(* PLC project Sin nombre, Desconocido Sin nombre 1 *)
(* stored: creationDateTime 2024-04-02T14:40:19, modificationDateTime 2024-04-04T08:12:00 *)

PROGRAM program0
  VAR
    START AT %IX0.0 : BOOL;
    STOP AT %IX0.1 : BOOL;
    INPUT0 AT %IX0.2 : BOOL := TRUE;
    OUTPUT0 AT %QX0.0 : BOOL;
    OUTPUT1 AT %QX0.1 : BOOL;
    STOP_LIGHT AT %QX0.2 : BOOL;
    START_LIGHT AT %QX0.3 : BOOL;
  END_VAR
  VAR
    IR1 : BOOL;
    IR2 : BOOL;
    IR3 : BOOL;
    IR4 : BOOL;
    IR5 : BOOL;
    TON_TIME1 : TIME := T#5S;
    COUNT_START : INT := 5;
    TON0 : TON;
    CTU0 : CTU;
  END_VAR
  VAR  (* added by the conversion: wires and edge detectors of the diagram *)
    R_TRIG1 : R_TRIG;
  END_VAR

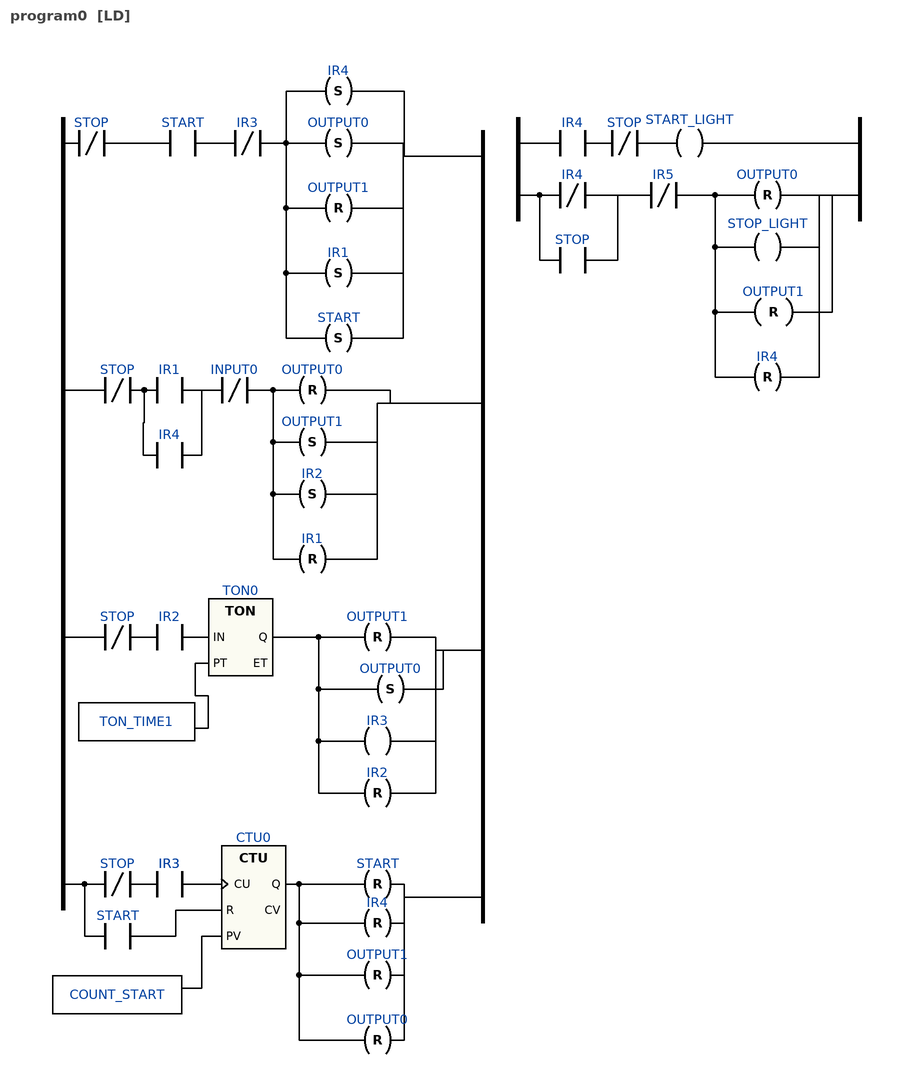
(* LD diagram, written out as Structured Text *)
IF NOT STOP AND START AND NOT IR3 THEN OUTPUT0 := TRUE; END_IF;
IF NOT STOP AND START AND NOT IR3 THEN OUTPUT1 := FALSE; END_IF;
IF NOT STOP AND START AND NOT IR3 THEN IR1 := TRUE; END_IF;
IF NOT STOP AND (IR1 OR IR4) AND NOT INPUT0 THEN OUTPUT0 := FALSE; END_IF;
IF NOT STOP AND (IR1 OR IR4) AND NOT INPUT0 THEN OUTPUT1 := TRUE; END_IF;
IF NOT STOP AND (IR1 OR IR4) AND NOT INPUT0 THEN IR2 := TRUE; END_IF;
TON0(IN := NOT STOP AND IR2, PT := TON_TIME1);
IF TON0.Q THEN OUTPUT0 := TRUE; END_IF;
IF TON0.Q THEN OUTPUT1 := FALSE; END_IF;
IR3 := TON0.Q;
R_TRIG1(CLK := NOT STOP AND IR3);
CTU0(CU := R_TRIG1.Q, R := START, PV := COUNT_START);
IF CTU0.Q THEN START := FALSE; END_IF;
START_LIGHT := IR4 AND NOT STOP;
STOP_LIGHT := (NOT IR4 OR STOP) AND NOT IR5;
IF CTU0.Q THEN OUTPUT1 := FALSE; END_IF;
IF CTU0.Q THEN OUTPUT0 := FALSE; END_IF;
IF NOT STOP AND START AND NOT IR3 THEN START := TRUE; END_IF;
IF (NOT IR4 OR STOP) AND NOT IR5 THEN OUTPUT0 := FALSE; END_IF;
IF (NOT IR4 OR STOP) AND NOT IR5 THEN OUTPUT1 := FALSE; END_IF;
IF NOT STOP AND START AND NOT IR3 THEN IR4 := TRUE; END_IF;
IF CTU0.Q THEN IR4 := FALSE; END_IF;
IF (NOT IR4 OR STOP) AND NOT IR5 THEN IR4 := FALSE; END_IF;
IF TON0.Q THEN IR2 := FALSE; END_IF;
IF NOT STOP AND (IR1 OR IR4) AND NOT INPUT0 THEN IR1 := FALSE; END_IF;
(* drawn but not wired to any output: IR3 *)
END_PROGRAM

CONFIGURATION Config0
  RESOURCE Res0 ON PLC
    TASK task0(INTERVAL := T#20ms, PRIORITY := 0);
    PROGRAM instance0 WITH task0 : program0;
  END_RESOURCE
END_CONFIGURATION
